# EPICS autosave request: ipApp/Db/ADAM_4018_settings.req
$(P)$(R):read.SCAN
